SYSTEM TEST_SYS3 (* System Configuration for testing TEST_DEV2 *)
  (* Standard: 61499-1 *)
  (* Version 0.0, 2004-06-08, JHC, Rockwell Automation *)
  APPLICATION APP1
  END_APPLICATION
  DEVICE DEV1 : FRAME_DEVICE
    RESOURCE INPUTS : PANEL_RESOURCE
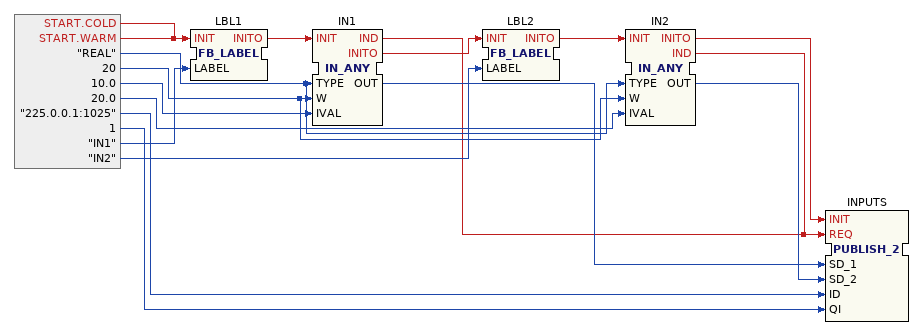
      FBS
        IN1 : IN_ANY;
        IN2 : IN_ANY;
        INPUTS : PUBLISH_2;
        LBL1 : FB_LABEL;
        LBL2 : FB_LABEL;
      END_FBS
      EVENT_CONNECTIONS
        IN2.INITO TO INPUTS.INIT;
        IN1.IND TO INPUTS.REQ;
        IN2.IND TO INPUTS.REQ;
        START.COLD TO LBL1.INIT;
        START.WARM TO LBL1.INIT;
        LBL1.INITO TO IN1.INIT;
        IN1.INITO TO LBL2.INIT;
        LBL2.INITO TO IN2.INIT;
      END_CONNECTIONS
      DATA_CONNECTIONS
        IN1.OUT TO INPUTS.SD_1;
        IN2.OUT TO INPUTS.SD_2;
        "REAL" TO IN1.TYPE;
        "REAL" TO IN2.TYPE;
        20 TO IN1.W;
        20 TO IN2.W;
        10.0 TO IN1.IVAL;
        20.0 TO IN2.IVAL;
        "225.0.0.1:1025" TO INPUTS.ID;
        1 TO INPUTS.QI;
        "IN1" TO LBL1.LABEL;
        "IN2" TO LBL2.LABEL;
      END_CONNECTIONS
    END_RESOURCE
    RESOURCE OUTPUTS : PANEL_RESOURCE
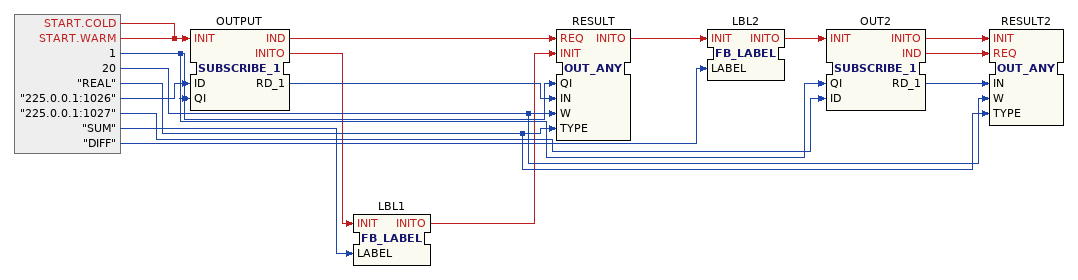
      FBS
        OUTPUT : SUBSCRIBE_1;
        RESULT : OUT_ANY;
        OUT2 : SUBSCRIBE_1;
        RESULT2 : OUT_ANY;
        LBL1 : FB_LABEL;
        LBL2 : FB_LABEL;
      END_FBS
      EVENT_CONNECTIONS
        START.COLD TO OUTPUT.INIT;
        START.WARM TO OUTPUT.INIT;
        OUTPUT.IND TO RESULT.REQ;
        OUT2.INITO TO RESULT2.INIT;
        OUT2.IND TO RESULT2.REQ;
        OUTPUT.INITO TO LBL1.INIT;
        LBL1.INITO TO RESULT.INIT;
        RESULT.INITO TO LBL2.INIT;
        LBL2.INITO TO OUT2.INIT;
      END_CONNECTIONS
      DATA_CONNECTIONS
        1 TO RESULT.QI;
        OUTPUT.RD_1 TO RESULT.IN;
        20 TO RESULT.W;
        "REAL" TO RESULT.TYPE;
        "225.0.0.1:1026" TO OUTPUT.ID;
        1 TO OUTPUT.QI;
        1 TO OUT2.QI;
        "225.0.0.1:1027" TO OUT2.ID;
        OUT2.RD_1 TO RESULT2.IN;
        20 TO RESULT2.W;
        "REAL" TO RESULT2.TYPE;
        "SUM" TO LBL1.LABEL;
        "DIFF" TO LBL2.LABEL;
      END_CONNECTIONS
    END_RESOURCE
  END_DEVICE
  DEVICE DEV2 : TEST_DEV2
    RESOURCE RES1 : TEST_RES2
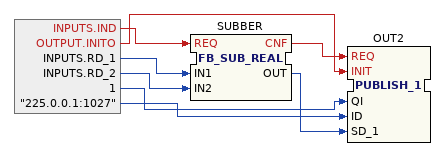
      FBS
        SUBBER : FB_SUB_REAL;
        OUT2 : PUBLISH_1;
      END_FBS
      EVENT_CONNECTIONS
        INPUTS.IND TO SUBBER.REQ;
        SUBBER.CNF TO OUT2.REQ;
        OUTPUT.INITO TO OUT2.INIT;
      END_CONNECTIONS
      DATA_CONNECTIONS
        INPUTS.RD_1 TO SUBBER.IN1;
        INPUTS.RD_2 TO SUBBER.IN2;
        1 TO OUT2.QI;
        "225.0.0.1:1027" TO OUT2.ID;
        SUBBER.OUT TO OUT2.SD_1;
      END_CONNECTIONS
    END_RESOURCE
  END_DEVICE
  DATA_CONNECTIONS (* parameter values *)
    [2,1] TO DEV1.GRID;
    [100,100,225,150] TO DEV1.BOUNDS;
  END_CONNECTIONS
END_SYSTEM
